INTERFACE I_SR1000

END_INTERFACE

(* stored: Version 1.1.0.1, ProductVersion 3.1.4024.6
   Itf I_SR1000: Id {db3901d9-9665-4496-bd15-9552792e4770} *)
